// TIA Portal V20 export
// export: Created 2026-04-11T06:02:30.0116196Z, ExportSetting WithDefaults, DisplayName Totally Integrated Automation Portal, DisplayVersion V20, DisplayName TIA Portal Openness, DisplayVersion V20, DisplayName TIA Portal Version Control Interface, DisplayVersion V20, DisplayName STEP 7 Professional, DisplayVersion V20, DisplayName STEP 7 Safety, DisplayVersion V20, DisplayName WinCC Basic/Comfort/Advanced, DisplayVersion V20, DisplayName WinCC Unified, DisplayVersion V20
TYPE "udtError_SoftStarter"
// stored: IsFailsafeCompliant false
   STRUCT
      NoSignalOnRun { ExternalWritable := 'False'} : Bool;   // No on/run signal from sof t starter
      NoSignalBypass { ExternalWritable := 'False'} : Bool;   // No bypass signal from soft starter
      MotorNotStopped { ExternalWritable := 'False'} : Bool;   // Soft starter doesn't stop
      SoftStarterFault { ExternalWritable := 'False'} : Bool;   // Overload or general fault from soft starter module
      SoftStarterWarning { ExternalWritable := 'False'} : Bool;   // General warning from soft starter module
      MotorProtectorTripped { ExternalWritable := 'False'} : Bool;   // Motor protector tripped
      LocalDisconnectOff { ExternalWritable := 'False'} : Bool;   // Local disconnect off
      DeviceNotReady { ExternalWritable := 'False'} : Bool;   // No Ready signal from soft starter
   END_STRUCT;
END_TYPE
